FUNCTION_BLOCK FB_XV03_DiagnosisParser_Tests EXTENDS FB_TestSuite
VAR_INPUT
END_VAR
VAR_OUTPUT
END_VAR
VAR
	_parser	: FB_XV03_DiagnosticsParser;
END_VAR

END_FUNCTION_BLOCK

(* stored: Version 1.1.0.1, ProductVersion 3.1.4024.13
   POU FB_XV03_DiagnosisParser_Tests: Id {484a256a-2e71-01b4-00e0-7b3512b39520}, SpecialFunc None *)
